// TIA Portal project "Trabalho automação" (V17)
// Vorlageprojekt für das Buch mit Zielsystem S7-1200

(* hardware
DEVICE "S7-1200-Station_1"  S7-1200 Station
   slot 0: "Baugruppenträger_0"  Rack  V1.0
   slot 1: "PLC_1"  CPU 1211C DC/DC/DC  6ES7 211-1AE40-0XB0  V4.1
*)

// ===== PLC "PLC_1"  CPU 1211C DC/DC/DC =====

VAR_GLOBAL   // PLC tag table "Standard-Variablentabelle"
   "At exit" AT %I0.0 : Bool;
   "Start" AT %I0.1 : Bool;
   "Reset" AT %I0.2 : Bool;
   "Stop" AT %I0.3 : Bool;
   "Emergency stop" AT %I0.4 : Bool;
   "Auto" AT %I0.5 : Bool;
   "Manual" AT %I0.6 : Bool;
   "Entry conveyor" AT %Q0.0 : Bool;
   "Stop blade" AT %Q0.1 : Bool;
   "Exit conveyor" AT %Q0.2 : Bool;
   "Sorter 1 turn" AT %Q0.3 : Bool;
   "Sorter 1 belt" AT %Q0.4 : Bool;
   "Sorter 2 turn" AT %Q0.5 : Bool;
   "Sorter 2 belt" AT %Q0.6 : Bool;
   "Sorter 3 turn" AT %Q0.7 : Bool;
   "Sorter 3 belt" AT %Q1.0 : Bool;
   "Start light" AT %Q1.1 : Bool;
   "Reset light" AT %Q1.2 : Bool;
   "Stop light" AT %Q1.3 : Bool;
   "Counter 1" AT %QD30 : DInt;
   "Counter 2" AT %QD34 : DInt;
   "Counter 3" AT %QD38 : DInt;
   "Vision sensor" AT %ID30 : DInt;
   "Digital output Byte 0" AT %QB0 : Byte;
   "Digital output Byte 1" AT %QB1 : Byte;
   "Clock_byte" AT %MB0 : Byte;
   "Clock_10Hz" AT %M0.0 : Bool;
   "Clock_5Hz" AT %M0.1 : Bool;
   "Clock_2.5Hz" AT %M0.2 : Bool;
   "Clock_2Hz" AT %M0.3 : Bool;
   "Clock_1.25Hz" AT %M0.4 : Bool;
   "Clock_1Hz" AT %M0.5 : Bool;
   "Clock_0.625Hz" AT %M0.6 : Bool;
   "Clock_0.5Hz" AT %M0.7 : Bool;
END_VAR

DATA_BLOCK "DB"   // DB2
{ S7_Optimized_Access := 'TRUE' }
VERSION : 0.1
   VAR
      Manual_cicle : Bool;
      condition : Int;
      End_cond_1 : Bool;
      End_cond_2 : Bool;
      End_cond_3 : Bool;
      Block_cicle : Bool;
      "M" : Array[0..4] of Bool;
      sts : Array[0..7] of Bool;
      Auto_cicle : Bool;
      Enable : Bool;
   END_VAR
BEGIN
END_DATA_BLOCK

// folder: System blocks/Program resources

DATA_BLOCK "IEC_Timer_0_DB"   // DB1
{ S7_Optimized_Access := 'TRUE' }
AUTHOR : Simatic
FAMILY : IEC
NAME : IEC_TMR
VERSION : 1.0
// stored: InstanceOfName IEC_TIMER
"IEC_TIMER"
BEGIN
END_DATA_BLOCK

DATA_BLOCK "IEC_Timer_2_DB"   // DB3
{ S7_Optimized_Access := 'TRUE' }
AUTHOR : Simatic
FAMILY : IEC
NAME : IEC_TMR
VERSION : 1.0
// stored: InstanceOfName IEC_TIMER
"IEC_TIMER"
BEGIN
END_DATA_BLOCK

DATA_BLOCK "IEC_Timer_3_DB"   // DB4
{ S7_Optimized_Access := 'TRUE' }
AUTHOR : Simatic
FAMILY : IEC
NAME : IEC_TMR
VERSION : 1.0
// stored: InstanceOfName IEC_TIMER
"IEC_TIMER"
BEGIN
END_DATA_BLOCK

DATA_BLOCK "IEC_Timer_4_DB"   // DB6
{ S7_Optimized_Access := 'TRUE' }
AUTHOR : Simatic
FAMILY : IEC
NAME : IEC_TMR
VERSION : 1.0
// stored: InstanceOfName IEC_TIMER
"IEC_TIMER"
BEGIN
END_DATA_BLOCK

DATA_BLOCK "IEC_Timer_5_DB"   // DB7
{ S7_Optimized_Access := 'TRUE' }
AUTHOR : Simatic
FAMILY : IEC
NAME : IEC_TMR
VERSION : 1.0
// stored: InstanceOfName IEC_TIMER
"IEC_TIMER"
BEGIN
END_DATA_BLOCK

DATA_BLOCK "IEC_Timer_6_DB"   // DB8
{ S7_Optimized_Access := 'TRUE' }
AUTHOR : Simatic
FAMILY : IEC
NAME : IEC_TMR
VERSION : 1.0
// stored: InstanceOfName IEC_TIMER
"IEC_TIMER"
BEGIN
END_DATA_BLOCK

DATA_BLOCK "IEC_Counter_0_DB"   // DB9
{ S7_Optimized_Access := 'TRUE' }
AUTHOR : Simatic
FAMILY : IEC
NAME : CNTR
VERSION : 1.0
// stored: InstanceOfName IEC_COUNTER
"IEC_COUNTER"
BEGIN
END_DATA_BLOCK

DATA_BLOCK "IEC_Timer_7_DB"   // DB10
{ S7_Optimized_Access := 'TRUE' }
AUTHOR : Simatic
FAMILY : IEC
NAME : IEC_TMR
VERSION : 1.0
// stored: InstanceOfName IEC_TIMER
"IEC_TIMER"
BEGIN
END_DATA_BLOCK

DATA_BLOCK "IEC_Timer_8_DB"   // DB11
{ S7_Optimized_Access := 'TRUE' }
AUTHOR : Simatic
FAMILY : IEC
NAME : IEC_TMR
VERSION : 1.0
// stored: InstanceOfName IEC_TIMER
"IEC_TIMER"
BEGIN
END_DATA_BLOCK

DATA_BLOCK "IEC_Counter_1_DB"   // DB12
{ S7_Optimized_Access := 'TRUE' }
AUTHOR : Simatic
FAMILY : IEC
NAME : CNTR
VERSION : 1.0
// stored: InstanceOfName IEC_COUNTER
"IEC_COUNTER"
BEGIN
END_DATA_BLOCK

DATA_BLOCK "IEC_Timer_9_DB"   // DB13
{ S7_Optimized_Access := 'TRUE' }
AUTHOR : Simatic
FAMILY : IEC
NAME : IEC_TMR
VERSION : 1.0
// stored: InstanceOfName IEC_TIMER
"IEC_TIMER"
BEGIN
END_DATA_BLOCK

DATA_BLOCK "IEC_Timer_10_DB"   // DB14
{ S7_Optimized_Access := 'TRUE' }
AUTHOR : Simatic
FAMILY : IEC
NAME : IEC_TMR
VERSION : 1.0
// stored: InstanceOfName IEC_TIMER
"IEC_TIMER"
BEGIN
END_DATA_BLOCK

DATA_BLOCK "IEC_Counter_2_DB"   // DB15
{ S7_Optimized_Access := 'TRUE' }
AUTHOR : Simatic
FAMILY : IEC
NAME : CNTR
VERSION : 1.0
// stored: InstanceOfName IEC_COUNTER
"IEC_COUNTER"
BEGIN
END_DATA_BLOCK

// folder: (top level)

FUNCTION "MHJ-PLC-Lab-Function-S71200" : Void   // FC9000, SCL
{ S7_Optimized_Access := 'TRUE' }
VERSION : 0.1
   VAR_TEMP
      rdTimeReturn : Int;
      outputTime : DTL;
      SyncVal : Byte;
      forVal : Int;
      forVal_2 : Int;
      Value : Byte;
   END_VAR
   VAR CONSTANT
      CompVal : Byte := 16#34;
      Value_01 : Byte := 16#11;
      Value_01_DW : DWord := 16#A165_D992;
      Value_02_DW : DWord := 16#58BE_4401;
   END_VAR
BEGIN

   #Value:=PEEK(area := 16#82,
        dbNumber := 0,
        byteOffset := 511);
   #Value := #Value + 1;

   POKE(area := 16#82,
        dbNumber := 0,
        byteOffset := 511,
        value := #Value);

   POKE(area:=16#81,
        dbNumber:=0,
        byteOffset:=1016,
        value:=#Value_01_DW);
   POKE(area := 16#81,
        dbNumber := 0,
        byteOffset := 1020,
        value := #Value_02_DW);

   POKE(area := 16#81,
        dbNumber := 0,
        byteOffset := 511,
        value := B#16#00);

   FOR #forVal := 0 TO 120 DO
       FOR #forVal_2:=0 TO 10 DO
           #rdTimeReturn:=RD_SYS_T(#outputTime);
           #rdTimeReturn := WR_SYS_T(#outputTime);
           #rdTimeReturn := RD_SYS_T(#outputTime);
           #rdTimeReturn := WR_SYS_T(#outputTime);
       END_FOR;
       #SyncVal:= PEEK(area := 16#81,
                      dbNumber := 0,
                      byteOffset := 511);
       IF #SyncVal = #CompVal THEN
          GOTO M_1;
       END_IF;
   END_FOR;
   RETURN;

   M_1:
   POKE(area := 16#81,
        dbNumber := 0,
        byteOffset := 511,
        value := B#16#0);
END_FUNCTION

ORGANIZATION_BLOCK "Main"   // OB1, LAD, ProgramCycle
TITLE = "Main Program Sweep (Cycle)"
{ S7_Optimized_Access := 'TRUE' }
VERSION : 0.1
   VAR_INPUT
      Initial_Call : Bool;   // Initial call of this OB
      Remanence : Bool;   // =True, if remanent data are available
   END_VAR
   VAR_TEMP   // added for the SCL form of the ladder/FBD networks
      _w1 : Bool;
      _w2 : Bool;
      _w3 : Bool;
      _w4 : Bool;
   END_VAR
BEGIN

REGION Network 1: Konnektierungsbaustein für PLC-Lab
   // Im Netzwerk 1 wird der Konnektierungsbaustein für PLC-Lab aufgerufen.
   // Dieser Aufruf darf nicht entfernt werden!
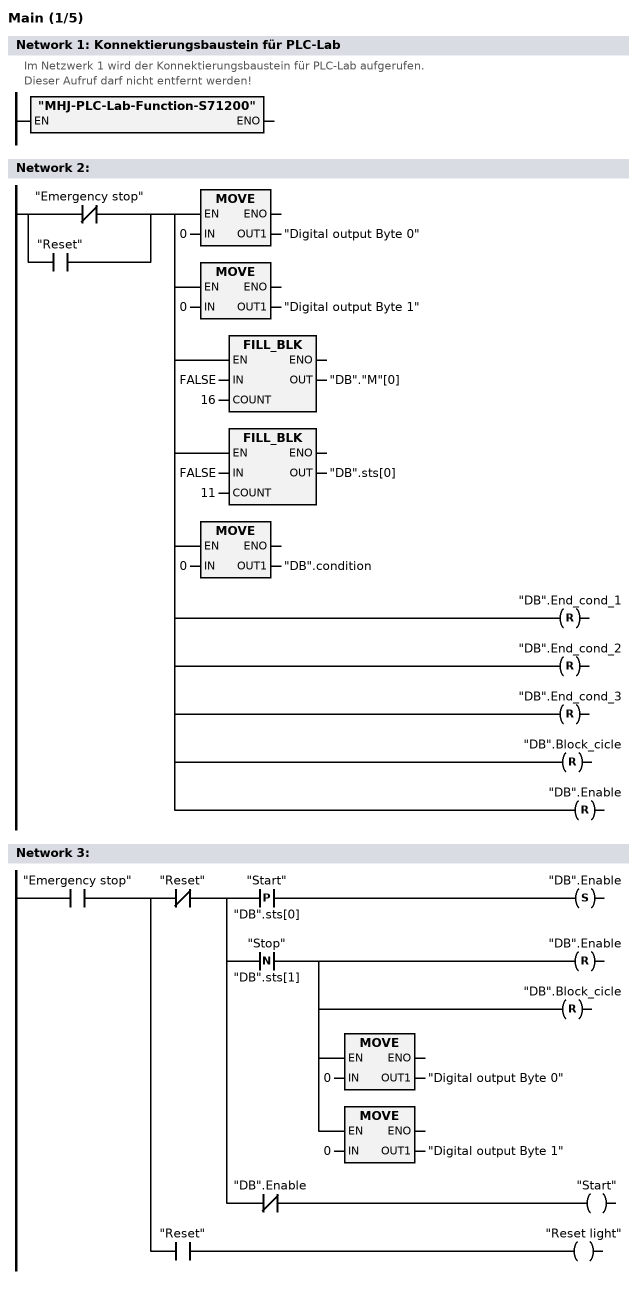
   RUNG wire#powerrail
      "MHJ-PLC-Lab-Function-S71200"()
   END_RUNG
   // the same network as SCL:
   "MHJ-PLC-Lab-Function-S71200"();
END_REGION

REGION Network 2
   RUNG wire#powerrail
      I_Contact( "Emergency stop" )
      wire#w1
      Move(in := 0, out1 => "Digital output Byte 0")
   END_RUNG
   RUNG wire#powerrail
      Contact( "Reset" )
   END_RUNG wire#w1
   RUNG wire#w1
      Move(in := 0, out1 => "Digital output Byte 1")
   END_RUNG
   RUNG wire#w1
      FillBlockI(in := FALSE, count := 16, out => "DB"."M"[0])
   END_RUNG
   RUNG wire#w1
      FillBlockI(in := FALSE, count := 11, out => "DB".sts[0])
   END_RUNG
   RUNG wire#w1
      Move(in := 0, out1 => "DB".condition)
   END_RUNG
   RUNG wire#w1
      R_Coil( "DB".End_cond_1 )
   END_RUNG
   RUNG wire#w1
      R_Coil( "DB".End_cond_2 )
   END_RUNG
   RUNG wire#w1
      R_Coil( "DB".End_cond_3 )
   END_RUNG
   RUNG wire#w1
      R_Coil( "DB".Block_cicle )
   END_RUNG
   RUNG wire#w1
      R_Coil( "DB".Enable )
   END_RUNG
   // the same network as SCL:
   IF NOT "Emergency stop" OR "Reset" THEN
       "Digital output Byte 0" := 0;
       "Digital output Byte 1" := 0;
   END_IF;
   #_w1 := NOT "Emergency stop" OR "Reset";
   IF #_w1 THEN
       FILL_BLK(IN := FALSE, COUNT := 16, OUT => "DB"."M"[0]);
       FILL_BLK(IN := FALSE, COUNT := 11, OUT => "DB".sts[0]);
       "DB".condition := 0;
       "DB".End_cond_1 := FALSE;
       "DB".End_cond_2 := FALSE;
       "DB".End_cond_3 := FALSE;
       "DB".Block_cicle := FALSE;
       "DB".Enable := FALSE;
   END_IF;
END_REGION

REGION Network 3
   RUNG wire#powerrail
      Contact( "Emergency stop" )
      wire#w1
      I_Contact( "Reset" )
      wire#w2
      P_Contact(operand := "Start", bit := "DB".sts[0])
      S_Coil( "DB".Enable )
   END_RUNG
   RUNG wire#w2
      N_Contact(operand := "Stop", bit := "DB".sts[1])
      wire#w3
      R_Coil( "DB".Enable )
   END_RUNG
   RUNG wire#w3
      R_Coil( "DB".Block_cicle )
   END_RUNG
   RUNG wire#w3
      Move(in := 0, out1 => "Digital output Byte 0")
   END_RUNG
   RUNG wire#w3
      Move(in := 0, out1 => "Digital output Byte 1")
   END_RUNG
   RUNG wire#w2
      I_Contact( "DB".Enable )
      Coil( "Start" )
   END_RUNG
   RUNG wire#w1
      Contact( "Reset" )
      Coil( "Reset light" )
   END_RUNG
   // the same network as SCL:
   #_w1 := "Emergency stop" AND NOT "Reset";
   #_w2 := #_w1 AND "Start" AND NOT "DB".sts[0];   // rising edge of "Start"
   "DB".sts[0] := "Start";
   IF #_w2 THEN "DB".Enable := TRUE; END_IF;
   #_w3 := #_w1 AND NOT "Stop" AND "DB".sts[1];   // falling edge of "Stop"
   "DB".sts[1] := "Stop";
   IF #_w3 THEN
       "DB".Enable := FALSE;
       "DB".Block_cicle := FALSE;
       "Digital output Byte 0" := 0;
       "Digital output Byte 1" := 0;
   END_IF;
   "Start" := #_w1 AND NOT "DB".Enable;
   "Reset light" := "Emergency stop" AND "Reset";
END_REGION

REGION Network 4
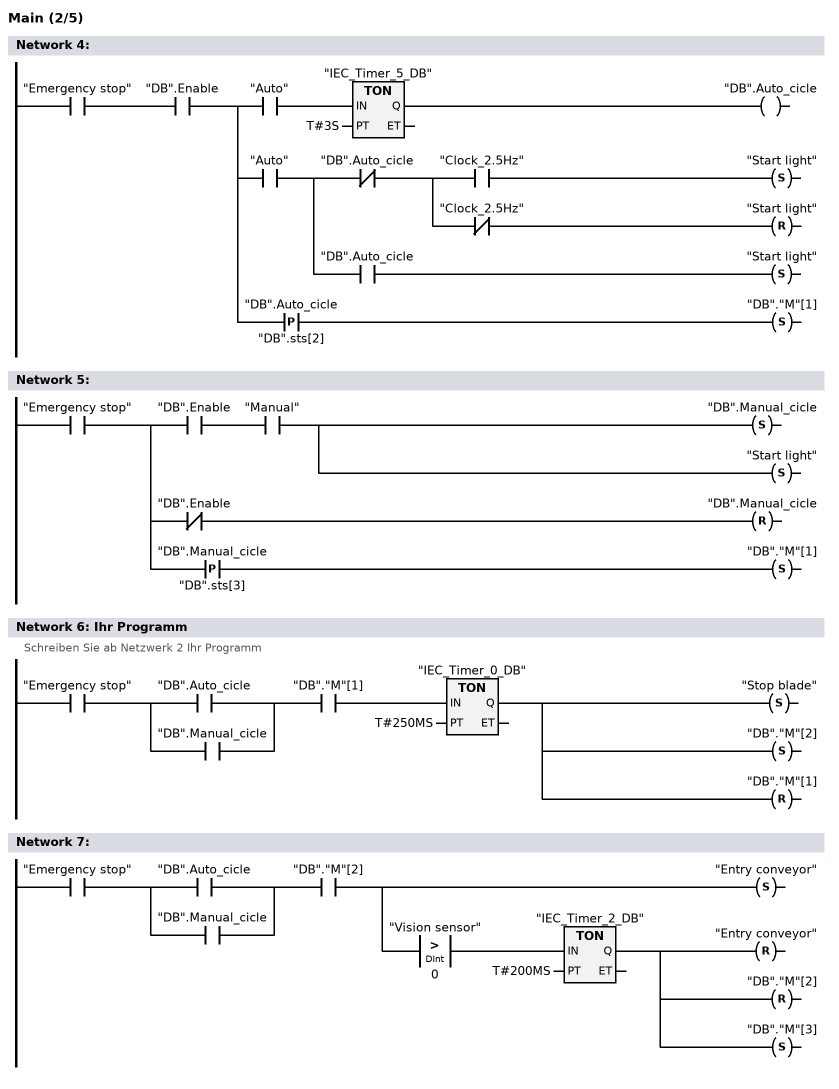
   #_w1 := "Emergency stop" AND "DB".Enable;
   "IEC_Timer_5_DB".TON(IN := #_w1 AND "Auto", PT := T#3S);
   "DB".Auto_cicle := "IEC_Timer_5_DB".Q;
   #_w2 := #_w1 AND "Auto";
   #_w3 := #_w2 AND NOT "DB".Auto_cicle;
   IF #_w3 AND "Clock_2.5Hz" THEN "Start light" := TRUE; END_IF;
   IF #_w3 AND NOT "Clock_2.5Hz" THEN "Start light" := FALSE; END_IF;
   IF #_w2 AND "DB".Auto_cicle THEN "Start light" := TRUE; END_IF;
   #_w4 := #_w1 AND "DB".Auto_cicle AND NOT "DB".sts[2];   // rising edge of "DB".Auto_cicle
   "DB".sts[2] := "DB".Auto_cicle;
   IF #_w4 THEN "DB"."M"[1] := TRUE; END_IF;
END_REGION

REGION Network 5
   RUNG wire#powerrail
      Contact( "Emergency stop" )
      wire#w1
      Contact( "DB".Enable )
      Contact( "Manual" )
      wire#w2
      S_Coil( "DB".Manual_cicle )
   END_RUNG
   RUNG wire#w2
      S_Coil( "Start light" )
   END_RUNG
   RUNG wire#w1
      I_Contact( "DB".Enable )
      R_Coil( "DB".Manual_cicle )
   END_RUNG
   RUNG wire#w1
      P_Contact(operand := "DB".Manual_cicle, bit := "DB".sts[3])
      S_Coil( "DB"."M"[1] )
   END_RUNG
   // the same network as SCL:
   IF "Emergency stop" AND "DB".Enable AND "Manual" THEN
       "DB".Manual_cicle := TRUE;
       "Start light" := TRUE;
   END_IF;
   IF "Emergency stop" AND NOT "DB".Enable THEN "DB".Manual_cicle := FALSE; END_IF;
   #_w1 := "Emergency stop" AND "DB".Manual_cicle AND NOT "DB".sts[3];   // rising edge of "DB".Manual_cicle
   "DB".sts[3] := "DB".Manual_cicle;
   IF #_w1 THEN "DB"."M"[1] := TRUE; END_IF;
END_REGION

REGION Network 6: Ihr Programm
   // Schreiben Sie ab Netzwerk 2 Ihr Programm
   "IEC_Timer_0_DB".TON(IN := "Emergency stop" AND ("DB".Auto_cicle OR "DB".Manual_cicle) AND "DB"."M"[1],
                        PT := T#250MS);
   IF "IEC_Timer_0_DB".Q THEN
       "Stop blade" := TRUE;
       "DB"."M"[2] := TRUE;
       "DB"."M"[1] := FALSE;
   END_IF;
END_REGION

REGION Network 7
   #_w1 := "Emergency stop" AND ("DB".Auto_cicle OR "DB".Manual_cicle) AND "DB"."M"[2];
   IF #_w1 THEN "Entry conveyor" := TRUE; END_IF;
   "IEC_Timer_2_DB".TON(IN := #_w1 AND ("Vision sensor" > 0), PT := T#200MS);
   IF "IEC_Timer_2_DB".Q THEN
       "Entry conveyor" := FALSE;
       "DB"."M"[2] := FALSE;
       "DB"."M"[3] := TRUE;
   END_IF;
END_REGION

REGION Network 8
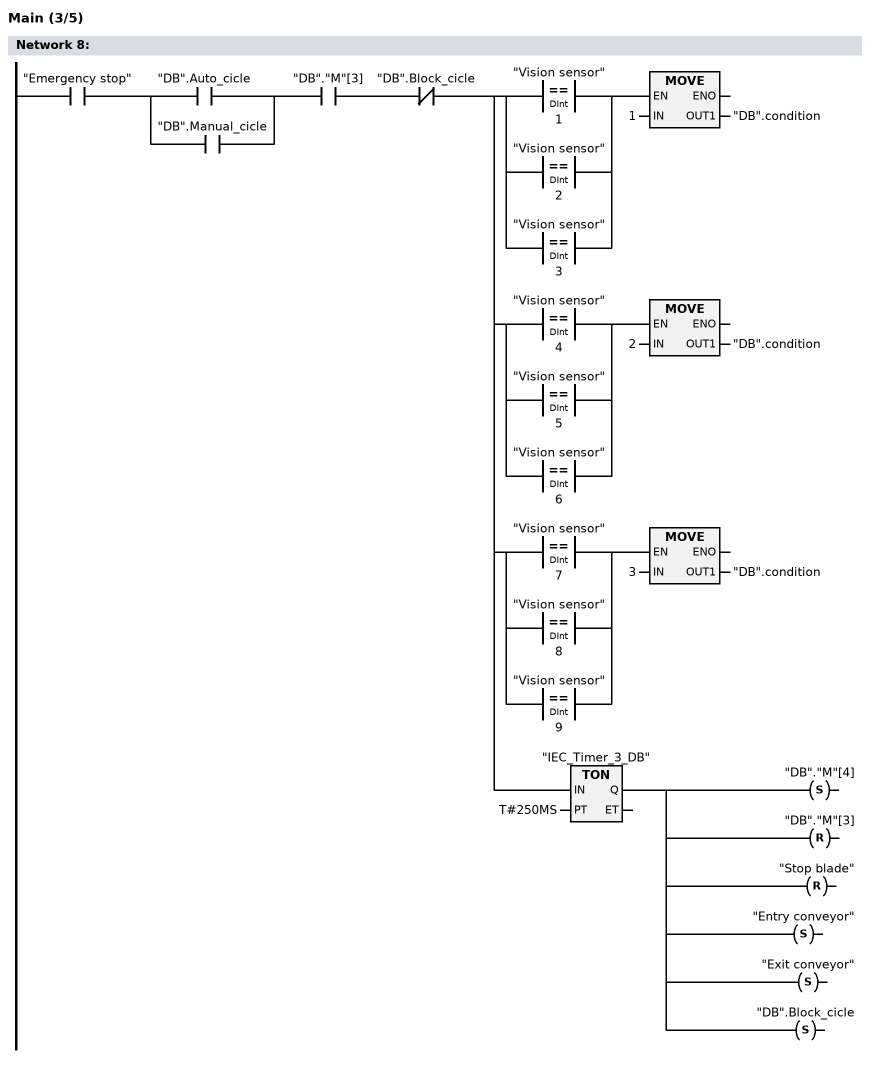
   #_w1 := "Emergency stop" AND ("DB".Auto_cicle OR "DB".Manual_cicle) AND "DB"."M"[3] AND NOT "DB".Block_cicle;
   IF #_w1 AND (("Vision sensor" = 1) OR ("Vision sensor" = 2) OR ("Vision sensor" = 3)) THEN
       "DB".condition := 1;
   END_IF;
   IF #_w1 AND (("Vision sensor" = 4) OR ("Vision sensor" = 5) OR ("Vision sensor" = 6)) THEN
       "DB".condition := 2;
   END_IF;
   IF #_w1 AND (("Vision sensor" = 7) OR ("Vision sensor" = 8) OR ("Vision sensor" = 9)) THEN
       "DB".condition := 3;
   END_IF;
   "IEC_Timer_3_DB".TON(IN := #_w1, PT := T#250MS);
   IF "IEC_Timer_3_DB".Q THEN
       "DB"."M"[4] := TRUE;
       "DB"."M"[3] := FALSE;
       "Stop blade" := FALSE;
       "Entry conveyor" := TRUE;
       "Exit conveyor" := TRUE;
       "DB".Block_cicle := TRUE;
   END_IF;
END_REGION

REGION Network 9
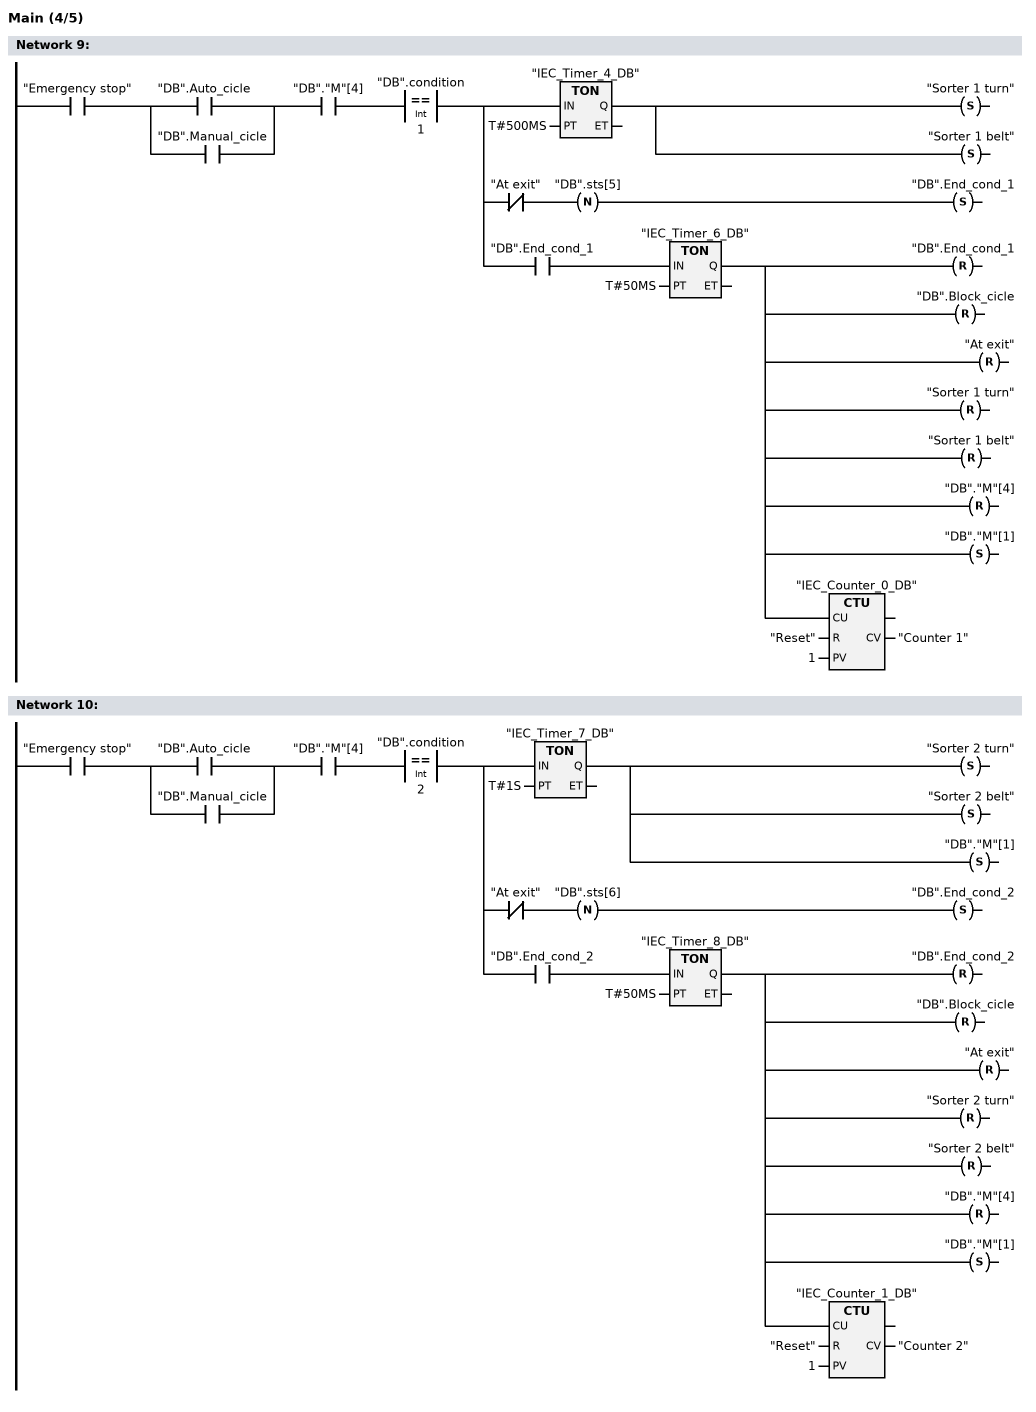
   #_w1 := "Emergency stop" AND ("DB".Auto_cicle OR "DB".Manual_cicle) AND "DB"."M"[4] AND ("DB".condition = 1);
   "IEC_Timer_4_DB".TON(IN := #_w1, PT := T#500MS);
   IF "IEC_Timer_4_DB".Q THEN
       "Sorter 1 turn" := TRUE;
       "Sorter 1 belt" := TRUE;
   END_IF;
   #_w2 := #_w1 AND NOT "At exit";
   #_w3 := NOT #_w2 AND "DB".sts[5];   // falling edge
   "DB".sts[5] := #_w2;
   IF #_w3 THEN "DB".End_cond_1 := TRUE; END_IF;
   "IEC_Timer_6_DB".TON(IN := #_w1 AND "DB".End_cond_1, PT := T#50MS);
   IF "IEC_Timer_6_DB".Q THEN
       "DB".End_cond_1 := FALSE;
       "DB".Block_cicle := FALSE;
       "At exit" := FALSE;
       "Sorter 1 turn" := FALSE;
       "Sorter 1 belt" := FALSE;
       "DB"."M"[4] := FALSE;
       "DB"."M"[1] := TRUE;
   END_IF;
   "IEC_Counter_0_DB".CTU(CU := "IEC_Timer_6_DB".Q, R := "Reset", PV := 1, CV => "Counter 1");
END_REGION

REGION Network 10
   #_w1 := "Emergency stop" AND ("DB".Auto_cicle OR "DB".Manual_cicle) AND "DB"."M"[4] AND ("DB".condition = 2);
   "IEC_Timer_7_DB".TON(IN := #_w1, PT := T#1S);
   IF "IEC_Timer_7_DB".Q THEN
       "Sorter 2 turn" := TRUE;
       "Sorter 2 belt" := TRUE;
       "DB"."M"[1] := TRUE;
   END_IF;
   #_w2 := #_w1 AND NOT "At exit";
   #_w3 := NOT #_w2 AND "DB".sts[6];   // falling edge
   "DB".sts[6] := #_w2;
   IF #_w3 THEN "DB".End_cond_2 := TRUE; END_IF;
   "IEC_Timer_8_DB".TON(IN := #_w1 AND "DB".End_cond_2, PT := T#50MS);
   IF "IEC_Timer_8_DB".Q THEN
       "DB".End_cond_2 := FALSE;
       "DB".Block_cicle := FALSE;
       "At exit" := FALSE;
       "Sorter 2 turn" := FALSE;
       "Sorter 2 belt" := FALSE;
       "DB"."M"[4] := FALSE;
       "DB"."M"[1] := TRUE;
   END_IF;
   "IEC_Counter_1_DB".CTU(CU := "IEC_Timer_8_DB".Q, R := "Reset", PV := 1, CV => "Counter 2");
END_REGION

REGION Network 11
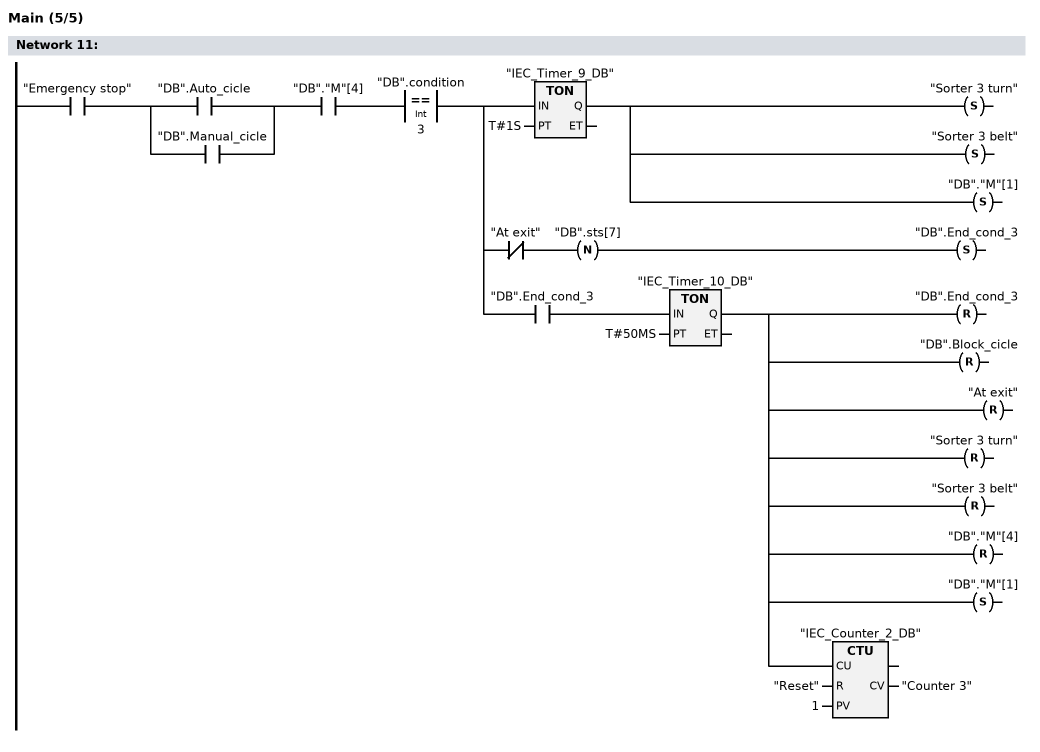
   #_w1 := "Emergency stop" AND ("DB".Auto_cicle OR "DB".Manual_cicle) AND "DB"."M"[4] AND ("DB".condition = 3);
   "IEC_Timer_9_DB".TON(IN := #_w1, PT := T#1S);
   IF "IEC_Timer_9_DB".Q THEN
       "Sorter 3 turn" := TRUE;
       "Sorter 3 belt" := TRUE;
       "DB"."M"[1] := TRUE;
   END_IF;
   #_w2 := #_w1 AND NOT "At exit";
   #_w3 := NOT #_w2 AND "DB".sts[7];   // falling edge
   "DB".sts[7] := #_w2;
   IF #_w3 THEN "DB".End_cond_3 := TRUE; END_IF;
   "IEC_Timer_10_DB".TON(IN := #_w1 AND "DB".End_cond_3, PT := T#50MS);
   IF "IEC_Timer_10_DB".Q THEN
       "DB".End_cond_3 := FALSE;
       "DB".Block_cicle := FALSE;
       "At exit" := FALSE;
       "Sorter 3 turn" := FALSE;
       "Sorter 3 belt" := FALSE;
       "DB"."M"[4] := FALSE;
       "DB"."M"[1] := TRUE;
   END_IF;
   "IEC_Counter_2_DB".CTU(CU := "IEC_Timer_10_DB".Q, R := "Reset", PV := 1, CV => "Counter 3");
END_REGION
END_ORGANIZATION_BLOCK